PROGRAM SlaveArmControl
VAR
	
	// all data from other tasks and controller 
	m_nullSlaveInputDataPool : ST_SlaveInputDataPool;
	
	// flag to init robot
	m_robotInit :BOOL :=FALSE;
	
	// wait time before robot init  for ethercat to be statble 
	m_robotInitWaitTime : LREAL:=0;
	
	// slave robot
	m_slaveRobot:FB_SlaveRobot;

	// code execute time measure
	m_codeTime : Profiler;
	
END_VAR

m_codeTime(START:=TRUE, RESET:=TRUE);

// wait communication to be stable
IF(m_robotInitWaitTime<g_robotInitWaitTime) THEN
	m_robotInitWaitTime := m_robotInitWaitTime+g_slaveArmCtrlCycleTime;
	RETURN;
END_IF

// robot init
IF m_robotInit =FALSE THEN
	m_slaveRobot.Init();
	m_robotInit:=TRUE;
END_IF

// robot run
m_slaveRobot.run(m_nullSlaveInputDataPool);

m_codeTime(START:=FALSE);

END_PROGRAM

(* stored: Version 1.1.0.1, ProductVersion 3.1.4024.12
   POU SlaveArmControl: Id {6192c11b-cd6e-4883-b627-958acfb9caf3}, SpecialFunc None *)
